FUNCTION TryConvert_UDINT_TO_LINT : BOOL
VAR_INPUT
	in : UDINT;
	out : REFERENCE TO LINT;
END_VAR

out := UDINT_TO_LINT(in);
TryConvert_UDINT_TO_LINT := TRUE;

END_FUNCTION

(* stored: Version 1.1.0.1, ProductVersion 3.1.4024.12
   POU TryConvert_UDINT_TO_LINT: Id {b7f07b39-b462-4822-91ff-2fa8a7ae22df}, SpecialFunc None *)
